TEXTLIST OutputText
  0 = 'OUT00 三色灯红' | Chinese: 'OUT00 三色灯红' | English: 'OUT00 Beacon_Red' | Vietnamese: 'OUT00 ?èn ?? ba màu ?'
  1 = 'OUT01 三色灯黄' | Chinese: 'OUT01 三色灯黄' | English: 'OUT01 Beacon_Yellow' | Vietnamese: 'OUT01 ?èn màu vàng ?'
  2 = 'OUT02 三色灯绿' | Chinese: 'OUT02 三色灯绿' | English: 'OUT02 Beacon_Green' | Vietnamese: 'OUT02 Màu xanh lá c?y ?èn ba màu ?'
  3 = 'OUT03 蜂鸣器' | Chinese: 'OUT03 蜂鸣器' | English: 'OUT03 Beacon_Buzzer' | Vietnamese: 'OUT03 buzzer ?'
  4 = 'OUT04 运行指示灯' | Chinese: 'OUT04 运行指示灯' | English: 'OUT04 Runing' | Vietnamese: 'OUT04 Ch?y ánh sáng ?'
  5 = 'OUT05 停止指示灯' | Chinese: 'OUT05 停止指示灯' | English: 'OUT05 Stop' | Vietnamese: 'OUT05 D?ng ?èn ?'
  6 = 'OUT06 照明灯' | Chinese: 'OUT06 照明灯' | English: 'OUT06 LED' | Vietnamese: 'OUT06 ?nh sáng ?'
  7 = 'OUT07 预留' | Chinese: 'OUT07 预留' | English: 'OUT07 None1' | Vietnamese: 'OUT07 Dành riêng ?'
  8 = 'OUT08 解锁站解压侧推气缸到原位' | Chinese: 'OUT08 解锁站解压侧推气缸到原位' | English: 'OUT08 OpenLockPressPush_Cyl_H' | Vietnamese: 'OUT08 OpenLockPressPush_Cyl_H'
  9 = 'OUT09 解锁站解压侧推气缸到工作位' | Chinese: 'OUT09 解锁站解压侧推气缸到工作位' | English: 'OUT09 OpenLockPressPush_Cyl_W' | Vietnamese: 'OUT09 OpenLockPressPush_Cyl_W'
  10 = 'OUT0A 解锁站解压旋转气缸到原位' | Chinese: 'OUT0A 解锁站解压旋转气缸到原位' | English: 'OUT0A OpenLockPressRotate_Cyl_H' | Vietnamese: 'OUT0A OpenLockPressRotate_Cyl_H'
  11 = 'OUT0B 解锁站解压旋转气缸到工作位' | Chinese: 'OUT0B 解锁站解压旋转气缸到工作位' | English: 'OUT0B OpenLockPressRotate_Cyl_W' | Vietnamese: 'OUT0B OpenLockPressRotate_Cyl_W'
  12 = 'OUT0C 主流线拨料升降气缸到原位' | Chinese: 'OUT0C 主流线拨料升降气缸到原位' | English: 'OUT0C Line0PushElevator_Cyl_H' | Vietnamese: 'OUT0C Line0PushElevator_Cyl_H'
  13 = 'OUT0D 主流线拨料升降气缸到工作位' | Chinese: 'OUT0D 主流线拨料升降气缸到工作位' | English: 'OUT0D Line0PushElevator_Cyl_W' | Vietnamese: 'OUT0D Line0PushElevator_Cyl_W'
  14 = 'OUT0E 接驳线前前阻挡气缸缩回' | Chinese: 'OUT0E 接驳线前前阻挡气缸缩回' | English: 'OUT0E AcquirePrevent2_Cyl_H' | Vietnamese: 'OUT0E AcquirePrevent2_Cyl_H'
  15 = 'OUT0F 接驳线前前阻挡气缸伸出' | Chinese: 'OUT0F 接驳线前前阻挡气缸伸出' | English: 'OUT0F AcquirePrevent2_Cyl_W' | Vietnamese: 'OUT0F AcquirePrevent2_Cyl_W'
  16 = 'OUT10 主流线分料气缸缩回' | Chinese: 'OUT10 主流线分料气缸缩回' | English: 'OUT10 Line0Part_Cyl_H' | Vietnamese: 'OUT10 Xi lanh c?a dòng chính rút lui ?'
  17 = 'OUT11 主流线分料气缸伸出' | Chinese: 'OUT11 主流线分料气缸伸出' | English: 'OUT11 Line0Part_Cyl_W' | Vietnamese: 'OUT11 Xi lanh dòng chính ra ngoài ?'
  18 = 'OUT12 主流线阻挡气缸缩回' | Chinese: 'OUT12 主流线阻挡气缸缩回' | English: 'OUT12 Line0Prevent_Cyl_H' | Vietnamese: 'OUT12 Dòng chính ng?n ch?n s? rút l?i c?a xi lanh ?'
  19 = 'OUT13 主流线阻挡气缸伸出' | Chinese: 'OUT13 主流线阻挡气缸伸出' | English: 'OUT13 Line0Prevent_Cyl_W' | Vietnamese: 'OUT13 Dòng chính ng?n các xi lanh thoát ra ?'
  20 = 'OUT14 主流线拨料气缸缩回' | Chinese: 'OUT14 主流线拨料气缸缩回' | English: 'OUT14 Line0Push_Cyl_H' | Vietnamese: 'OUT14 Xi lanh quay dòng chính rút lui ?'
  21 = 'OUT15 主流线拨料气缸伸出' | Chinese: 'OUT15 主流线拨料气缸伸出' | English: 'OUT15 Line0Push_Cyl_W' | Vietnamese: 'OUT15 Xi lanh cu?n dòng chính thò ra ?'
  22 = 'OUT16 接驳线前阻挡气缸缩回' | Chinese: 'OUT16 接驳线前阻挡气缸缩回' | English: 'OUT16 AcquirePrevent0_Cyl_H' | Vietnamese: 'OUT16 Khóa xi lanh tr??c d?y n?i rút l?i ?'
  23 = 'OUT17 接驳线前阻挡气缸伸出' | Chinese: 'OUT17 接驳线前阻挡气缸伸出' | English: 'OUT17 AcquirePrevent0_Cyl_W' | Vietnamese: 'OUT17 Ch?n xi lanh tr??c d?y n?i ?'
  24 = 'OUT18 接驳线后阻挡气缸缩回' | Chinese: 'OUT18 接驳线后阻挡气缸缩回' | English: 'OUT18 AcquirePrevent1_Cyl_H' | Vietnamese: 'OUT18 Khóa xi lanh l?i sau khi k?t n?i ?'
  25 = 'OUT19 接驳线后阻挡气缸伸出' | Chinese: 'OUT19 接驳线后阻挡气缸伸出' | English: 'OUT19 AcquirePrevent1_Cyl_W' | Vietnamese: 'OUT19 Ch?n xi lanh ra sau d?y n?i ?'
  26 = 'OUT1A 接驳线顶升气缸缩回' | Chinese: 'OUT1A 接驳线顶升气缸缩回' | English: 'OUT1A AcquireLift_Cyl_H' | Vietnamese: 'OUT1A Xi lanh n?ng d?y n?i rút l?i ?'
  27 = 'OUT1B 接驳线顶升气缸伸出' | Chinese: 'OUT1B 接驳线顶升气缸伸出' | English: 'OUT1B AcquireLift_Cyl_W' | Vietnamese: 'OUT1B Xi lanh c?m trên d?y d?n ra ngoài ?'
  28 = 'OUT1C 接驳模组拨料气缸缩回' | Chinese: 'OUT1C 接驳模组拨料气缸缩回' | English: 'OUT1C AcquirePush_Cyl_H' | Vietnamese: 'OUT1C Xi lanh k?t n?i m?-?un quay l?i ?'
  29 = 'OUT1D 接驳模组拨料气缸伸出' | Chinese: 'OUT1D 接驳模组拨料气缸伸出' | English: 'OUT1D AcquirePush_Cyl_W' | Vietnamese: 'OUT1D Xi lanh k?t n?i m?-?un phát ra ?'
  30 = 'OUT1E 接驳模组升降气缸缩回' | Chinese: 'OUT1E 接驳模组升降气缸缩回' | English: 'OUT1E AcquireElevator_Cyl_H' | Vietnamese: 'OUT1E Xi lanh n?ng m?-?un n?i rút l?i ?'
  31 = 'OUT1F 接驳模组升降气缸伸出' | Chinese: 'OUT1F 接驳模组升降气缸伸出' | English: 'OUT1F AcquireElevator_Cyl_W' | Vietnamese: 'OUT1F Xi lanh n?ng m?-?un n?i thò ra ?'
  32 = 'OUT20 转向站顶升气缸缩回' | Chinese: 'OUT20 转向站顶升气缸缩回' | English: 'OUT20 SteeringLift_Cyl_H' | Vietnamese: 'OUT20 Quay tr? l?i xi lanh ?'
  33 = 'OUT21 转向站顶升气缸伸出' | Chinese: 'OUT21 转向站顶升气缸伸出' | English: 'OUT21 SteeringLift_Cyl_W' | Vietnamese: 'OUT21 Các xi lanh m? ra ?'
  34 = 'OUT22 转向站接驳升降气缸缩回' | Chinese: 'OUT22 转向站接驳升降气缸缩回' | English: 'OUT22 SteeringAcquireElevator_Cyl_H' | Vietnamese: 'OUT22 Quay l?i v?i xi lanh n?ng t?i tr?m lái ?'
  35 = 'OUT23 转向站接驳升降气缸伸出' | Chinese: 'OUT23 转向站接驳升降气缸伸出' | English: 'OUT23 SteeringAcquireElevator_Cyl_W' | Vietnamese: 'OUT23 Các xi lanh n?ng ???c n?i v?i các tr?m r? ?'
  36 = 'OUT24 转向站旋转气缸缩回' | Chinese: 'OUT24 转向站旋转气缸缩回' | English: 'OUT24 SteeringRotate_Cyl_H' | Vietnamese: 'OUT24 Quay tr?m quay xi lanh ?? rút lui ?'
  37 = 'OUT25 转向站旋转气缸伸出' | Chinese: 'OUT25 转向站旋转气缸伸出' | English: 'OUT25 SteeringRotate_Cyl_W' | Vietnamese: 'OUT25 Các xi lanh xoay ? v? trí quay thò ra ?'
  38 = 'OUT26 转向站接驳限位气缸缩回' | Chinese: 'OUT26 转向站接驳限位气缸缩回' | English: 'OUT26 SteeringAcquireLimit_Cyl_H' | Vietnamese: 'OUT26 Quay l?i xi lanh gi?i h?n k?t n?i tr?m r? ?'
  39 = 'OUT27 转向站接驳限位气缸伸出' | Chinese: 'OUT27 转向站接驳限位气缸伸出' | English: 'OUT27 SteeringAcquireLimit_Cyl_W' | Vietnamese: 'OUT27 Xi lanh gi?i h?n k?t n?i v?i tr?m lái xe ???c thò ra ?'
  40 = 'OUT28 解锁站阻挡气缸缩回' | Chinese: 'OUT28 解锁站阻挡气缸缩回' | English: 'OUT28 OpenLockPrevent_Cyl_H' | Vietnamese: 'OUT28 Tr?m m? khóa ng?n ch?n s? rút lui xi lanh ?'
  41 = 'OUT29 解锁站阻挡气缸伸出' | Chinese: 'OUT29 解锁站阻挡气缸伸出' | English: 'OUT29 OpenLockPrevent_Cyl_W' | Vietnamese: 'OUT29 Tr?m m? khóa ng?n ch?n các xi lanh thò ra ?'
  42 = 'OUT2A 解锁站顶升气缸缩回' | Chinese: 'OUT2A 解锁站顶升气缸缩回' | English: 'OUT2A OpenLockLift_Cyl_H' | Vietnamese: 'OUT2A M? khóa tr?m n?ng xi lanh rút lui ?'
  43 = 'OUT2B 解锁站顶升气缸伸出' | Chinese: 'OUT2B 解锁站顶升气缸伸出' | English: 'OUT2B OpenLockLift_Cyl_W' | Vietnamese: 'OUT2B Xi lanh m? khóa tr? n?ng thò ra ?'
  44 = 'OUT2C 解锁站侧推气缸缩回' | Chinese: 'OUT2C 解锁站侧推气缸缩回' | English: 'OUT2C OpenLockPush_Cyl_H' | Vietnamese: 'OUT2C M? khóa các xi lanh ??y ga ?? rút lui ?'
  45 = 'OUT2D 解锁站侧推气缸伸出' | Chinese: 'OUT2D 解锁站侧推气缸伸出' | English: 'OUT2D OpenLockPush_Cyl_W' | Vietnamese: 'OUT2D M? khóa ga ??y xi lanh thò ra ?'
  46 = 'OUT2E 解锁站旋转气缸缩回' | Chinese: 'OUT2E 解锁站旋转气缸缩回' | English: 'OUT2E OpenLockRotate_Cyl_H' | Vietnamese: 'OUT2E M? khóa tr?m quay xi lanh rút lui ?'
  47 = 'OUT2F 解锁站旋转气缸伸出' | Chinese: 'OUT2F 解锁站旋转气缸伸出' | English: 'OUT2F OpenLockRotate_Cyl_W' | Vietnamese: 'OUT2F Xi lanh xoay ? v? trí m? khóa thò ra ?'
  48 = 'OUT30 解锁站侧推气缸2缩回' | Chinese: 'OUT30 解锁站侧推气缸2缩回' | English: 'OUT30 OpenLockPush2_Cyl_H' | Vietnamese: 'OUT30 M? khóa ga bên ??y xi lanh 2 rút lui ?'
  49 = 'OUT31 解锁站侧推气缸2伸出' | Chinese: 'OUT31 解锁站侧推气缸2伸出' | English: 'OUT31 OpenLockPush2_Cyl_W' | Vietnamese: 'OUT31 M? khóa ga ??y xi lanh 2 thò ra ?'
  50 = 'OUT32 取UC站阻挡气缸缩回' | Chinese: 'OUT32 取UC站阻挡气缸缩回' | English: 'OUT32 TakeUcPrevent_Cyl_H' | Vietnamese: 'OUT32 L?y các tr?m ng?n ch?n và rút l?i xi lanh ?'
  51 = 'OUT33 取UC站阻挡气缸伸出' | Chinese: 'OUT33 取UC站阻挡气缸伸出' | English: 'OUT33 TakeUcPrevent_Cyl_W' | Vietnamese: 'OUT33 L?y ga ng?n ch?n lít ra ?'
  52 = 'OUT34 取UC站顶升气缸缩回' | Chinese: 'OUT34 取UC站顶升气缸缩回' | English: 'OUT34 TakeUcLift_Cyl_H' | Vietnamese: 'OUT34 L?y xi lanh n?ng lên c?a tr?m UC và rút lui ?'
  53 = 'OUT35 取UC站顶升气缸伸出' | Chinese: 'OUT35 取UC站顶升气缸伸出' | English: 'OUT35 TakeUcLift_Cyl_W' | Vietnamese: 'OUT35 L?y xi lanh n?ng lên t? tr?m UC ?'
  54 = 'OUT36 取UC站侧推气缸缩回' | Chinese: 'OUT36 取UC站侧推气缸缩回' | English: 'OUT36 TakeUcPush_Cyl_H' | Vietnamese: 'OUT36 L?y xi lanh ??y bên tàu và rút lui ?'
  55 = 'OUT37 取UC站侧推气缸伸出' | Chinese: 'OUT37 取UC站侧推气缸伸出' | English: 'OUT37 TakeUcPush_Cyl_W' | Vietnamese: 'OUT37 L?y ga bên ??y ra kh?i xi lanh ?'
  56 = 'OUT38 取UC站旋转气缸缩回' | Chinese: 'OUT38 取UC站旋转气缸缩回' | English: 'OUT38 TakeUcRotate_Cyl_H' | Vietnamese: 'OUT38 L?y xi lanh quay ? tr?m UC và rút lui ?'
  57 = 'OUT39 取UC站旋转气缸伸出' | Chinese: 'OUT39 取UC站旋转气缸伸出' | English: 'OUT39 TakeUcRotate_Cyl_W' | Vietnamese: 'OUT39 L?y các xi lanh quay t? tr?m UC ?'
  58 = 'OUT3A 取UC站校平气缸原位' | Chinese: 'OUT3A 取UC站校平气缸原位' | English: 'OUT3A TakeUcStandard_Cyl_H' | Vietnamese: 'OUT3A L?y xi lanh ph?ng ? ga UC ?'
  59 = 'OUT3B 取UC站校平气缸工作位' | Chinese: 'OUT3B 取UC站校平气缸工作位' | English: 'OUT3B TakeUcStandard_Cyl_W' | Vietnamese: 'OUT3B Tr?m ki?m tra xi lanh b?ng ph?ng ?'
  60 = 'OUT3C 取UC站工装夹紧气缸原位' | Chinese: 'OUT3C 取UC站工装夹紧气缸原位' | English: 'OUT3C TakeUcFrockClamp_Cyl_H' | Vietnamese: 'OUT3C L?y xi lanh k?p vào v? trí c?a tr?m UC'
  61 = 'OUT3D 取UC站工装夹紧气缸工作位' | Chinese: 'OUT3D 取UC站工装夹紧气缸工作位' | English: 'OUT3D TakeUcFrockClamp_Cyl_W' | Vietnamese: 'OUT3D L?y v? trí làm vi?c xi lanh cài ??t ? ga UC'
  62 = 'OUT3E 下工装站阻挡气缸缩回' | Chinese: 'OUT3E 下工装站阻挡气缸缩回' | English: 'OUT3E UnloadFrockPrevent_Cyl_H' | Vietnamese: 'OUT3E Ng?n ch?n các xi lanh rút lui ?'
  63 = 'OUT3F 下工装站阻挡气缸伸出' | Chinese: 'OUT3F 下工装站阻挡气缸伸出' | English: 'OUT3F UnloadFrockPrevent_Cyl_W' | Vietnamese: 'OUT3F Ng?n ch?n các xi lanh ra ngoài ?'
  64 = 'OUT40 下工装站顶升气缸缩回' | Chinese: 'OUT40 下工装站顶升气缸缩回' | English: 'OUT40 UnloadFrockLift_Cyl_H' | Vietnamese: 'OUT40 Xi lanh n?ng xu?ng ga xu?ng rút lui ?'
  65 = 'OUT41 下工装站顶升气缸伸出' | Chinese: 'OUT41 下工装站顶升气缸伸出' | English: 'OUT41 UnloadFrockLift_Cyl_W' | Vietnamese: 'OUT41 Xi lanh n?ng lên t? tr?m t?i xu?ng ?'
  66 = 'OUT42 下工装站拨料气缸缩回' | Chinese: 'OUT42 下工装站拨料气缸缩回' | English: 'OUT42 UnloadFrockPush_Cyl_H' | Vietnamese: 'OUT42 Xi lanh xi lanh quay tr? l?i tr?m t?i xu?ng ?'
  67 = 'OUT43 下工装站拨料气缸伸出' | Chinese: 'OUT43 下工装站拨料气缸伸出' | English: 'OUT43 UnloadFrockPush_Cyl_W' | Vietnamese: 'OUT43 Xi lanh ngu?n l?c ti?p theo ?'
  68 = 'OUT44 取UC模组平移Y气缸缩回' | Chinese: 'OUT44 取UC模组平移Y气缸缩回' | English: 'OUT44 TakeUc1Y_Cyl_H' | Vietnamese: 'OUT44 L?y m?-?un UC chuy?n xi lanh Y và rút lui ?'
  69 = 'OUT45 取UC模组平移Y气缸伸出' | Chinese: 'OUT45 取UC模组平移Y气缸伸出' | English: 'OUT45 TakeUc1Y_Cyl_W' | Vietnamese: 'OUT45 L?y m?-?un UC và di chuy?n xi lanh Y ra ngoài ?'
  70 = 'OUT46 取UC模组升降Z1气缸缩回' | Chinese: 'OUT46 取UC模组升降Z1气缸缩回' | English: 'OUT46 TakeUc1Z1_Cyl_H' | Vietnamese: 'OUT46 L?y m?-?un UC n?ng xi lanh Z1 ?? rút lui ?'
  71 = 'OUT47 取UC模组升降Z1气缸伸出' | Chinese: 'OUT47 取UC模组升降Z1气缸伸出' | English: 'OUT47 TakeUc1Z1_Cyl_W' | Vietnamese: 'OUT47 N?ng xi lanh ra kh?i m?-?un UC ?'
  72 = 'OUT48 取UC模组升降Z2气缸缩回' | Chinese: 'OUT48 取UC模组升降Z2气缸缩回' | English: 'OUT48 TakeUc1Z2_Cyl_H' | Vietnamese: 'OUT48 L?y m?-?un UC n?ng xi lanh Z2 ?? rút lui ?'
  73 = 'OUT49 取UC模组升降Z2气缸伸出' | Chinese: 'OUT49 取UC模组升降Z2气缸伸出' | English: 'OUT49 TakeUc1Z2_Cyl_W' | Vietnamese: 'OUT49 ??a ?ng n?ng Z2 ra kh?i m?-?un UC ?'
  74 = 'OUT4A 取UC模组旋转气缸缩回' | Chinese: 'OUT4A 取UC模组旋转气缸缩回' | English: 'OUT4A TakeUc1Rotate_Cyl_H' | Vietnamese: 'OUT4A Thu h?i xi lanh quay b?ng m?-?un UC ?'
  75 = 'OUT4B 取UC模组旋转气缸伸出' | Chinese: 'OUT4B 取UC模组旋转气缸伸出' | English: 'OUT4B TakeUc1Rotate_Cyl_W' | Vietnamese: 'OUT4B L?y m?-?un UC xoay xi lanh ra ngoài ?'
  76 = 'OUT4C 取UC模组夹紧气缸缩回' | Chinese: 'OUT4C 取UC模组夹紧气缸缩回' | English: 'OUT4C TakeUc1Clamp_Cyl_H' | Vietnamese: 'OUT4C L?y m?-?un UC k?p xi lanh ?? rút lui ?'
  77 = 'OUT4D 取UC模组夹紧气缸伸出' | Chinese: 'OUT4D 取UC模组夹紧气缸伸出' | English: 'OUT4D TakeUc1Clamp_Cyl_W' | Vietnamese: 'OUT4D L?y m?-?un và k?p ?ng ra ?'
  78 = 'OUT4E 下UC皮带升降气缸缩回' | Chinese: 'OUT4E 下UC皮带升降气缸缩回' | English: 'OUT4E UnloadUcElevator_Cyl_H' | Vietnamese: 'OUT4E Thu h?i xi lanh n?ng d??i vành ?ai UC ?'
  79 = 'OUT4F 下UC皮带升降气缸伸出' | Chinese: 'OUT4F 下UC皮带升降气缸伸出' | English: 'OUT4F UnloadUcElevator_Cyl_W' | Vietnamese: 'OUT4F Xi lanh n?ng d??i vành ?ai UC thò ra ?'
  80 = 'OUT50 下UC皮带拨料气缸缩回' | Chinese: 'OUT50 下UC皮带拨料气缸缩回' | English: 'OUT50 UnloadUcConveyorPush_Cyl_H' | Vietnamese: 'OUT50 Quay l?i xi lanh quay d??i vành ?ai UC ?'
  81 = 'OUT51 下UC皮带拨料气缸伸出' | Chinese: 'OUT51 下UC皮带拨料气缸伸出' | English: 'OUT51 UnloadUcConveyorPush_Cyl_W' | Vietnamese: 'OUT51 Cái xi lanh d??i vành ?ai UC thò ra ?'
  82 = 'OUT52 下工装皮带升降气缸缩回' | Chinese: 'OUT52 下工装皮带升降气缸缩回' | English: 'OUT52 UnloadFrockConveyorPrevent_Cyl_H' | Vietnamese: 'OUT52 Th?t l?ng n?ng xi lanh kéo xu?ng ?'
  83 = 'OUT53 下工装皮带升降气缸伸出' | Chinese: 'OUT53 下工装皮带升降气缸伸出' | English: 'OUT53 UnloadFrockConveyorPrevent_Cyl_W' | Vietnamese: 'OUT53 Xi lanh n?ng vành ?ai c?ng vi?c thò ra ?'
  84 = 'OUT54 下工装皮带拨料气缸缩回' | Chinese: 'OUT54 下工装皮带拨料气缸缩回' | English: 'OUT54 UnloadFrockConveyorPush_Cyl_H' | Vietnamese: 'OUT54 ?óng gói vành ?ai xi lanh quay l?i ?'
  85 = 'OUT55 下工装皮带拨料气缸伸出' | Chinese: 'OUT55 下工装皮带拨料气缸伸出' | English: 'OUT55 UnloadFrockConveyorPush_Cyl_W' | Vietnamese: 'OUT55 Xi lanh vành ?ai c?ng c? thò ra ?'
  86 = 'OUT56 接驳线前步进' | Chinese: 'OUT56 接驳线前步进' | English: 'OUT56 AcquireFrontAxis' | Vietnamese: 'OUT56 AcquireFrontAxis'
  87 = 'OUT57 接驳线步进' | Chinese: 'OUT57 接驳线步进' | English: 'OUT57 AcquireAxis' | Vietnamese: 'OUT57 B??c trên d?y n?i ?'
  88 = 'OUT58 拆解线步进' | Chinese: 'OUT58 拆解线步进' | English: 'OUT58 DismantlingAxis' | Vietnamese: 'OUT58 B??c c?t d?y ?'
  89 = 'OUT59 下UC皮带步进' | Chinese: 'OUT59 下UC皮带步进' | English: 'OUT59 UnloadUcAxis' | Vietnamese: 'OUT59 B??c xu?ng d??i vành ?ai UC ?'
  90 = 'OUT5A 下工装皮带步进' | Chinese: 'OUT5A 下工装皮带步进' | English: 'OUT5A UnloadFrock' | Vietnamese: 'OUT5A D?y n?t di chuy?n ?'
  91 = 'OUT5B 预留' | Chinese: 'OUT5B 预留' | English: 'OUT5B None21' | Vietnamese: 'OUT5B Dành riêng ?'
  92 = 'OUT5C 下UC皮带翻转气缸缩回' | Chinese: 'OUT5C 下UC皮带翻转气缸缩回' | English: 'OUT5C UnloadUcBeltTipper_Cyl_H' | Vietnamese: 'OUT5C Quay ng??c xi lanh l?i ?'
  93 = 'OUT5D 下UC皮带翻转气缸伸出' | Chinese: 'OUT5D 下UC皮带翻转气缸伸出' | English: 'OUT5D UnloadUcBeltTipper_Cyl_W' | Vietnamese: 'OUT5D Cái xi lanh xoay d??i vành ?ai UC thò ra ?'
  94 = 'OUT5E 下UC皮带顶升气缸缩回' | Chinese: 'OUT5E 下UC皮带顶升气缸缩回' | English: 'OUT5E UnloadUcBeltLift_Cyl_H' | Vietnamese: 'OUT5E Co l?i xi lanh n?ng lên d??i vành ?ai UC ?'
  95 = 'OUT5F 下UC皮带顶升气缸伸出' | Chinese: 'OUT5F 下UC皮带顶升气缸伸出' | English: 'OUT5F UnloadUcBeltLift_Cyl_W' | Vietnamese: 'OUT5F Cái xi lanh n?ng lên d??i vành ?ai UC thò ra ?'
  96 = 'OUT60 解锁站升降气缸原位' | Chinese: 'OUT60 解锁站升降气缸原位' | English: 'OUT60 OpenLockElevator_Cyl_H' | Vietnamese: 'OUT60 M? khóa tr?m n?ng xi lanh v? trí ?'
  97 = 'OUT61 解锁站升降气缸工作位' | Chinese: 'OUT61 解锁站升降气缸工作位' | English: 'OUT61 OpenLockElevator_Cyl_W' | Vietnamese: 'OUT61 M? khóa tr?m n?ng xi lanh v? trí làm vi?c ?'
  98 = 'OUT62 解锁站解锁平移原位' | Chinese: 'OUT62 解锁站解锁平移原位' | English: 'OUT62 OpenLockTranslation_Cyl_H' | Vietnamese: 'OUT62 Tr?m m? khóa m? khóa chuy?n v? trí ?'
  99 = 'OUT63 解锁站解锁平移工作位' | Chinese: 'OUT63 解锁站解锁平移工作位' | English: 'OUT63 OpenLockTranslation_Cyl_W' | Vietnamese: 'OUT63 Tr?m m? khóa m? khóa chuy?n v? trí làm vi?c ?'
  100 = 'OUT64 解锁站按压气缸到原位' | Chinese: 'OUT64 解锁站按压气缸到原位' | English: 'OUT64 OpenLockPin_Cyl_H' | Vietnamese: 'OUT64 M? khóa tr?m nh?n xi lanh vào v? trí ?'
  101 = 'OUT65 解锁站按压气缸到工作位' | Chinese: 'OUT65 解锁站按压气缸到工作位' | English: 'OUT65 OpenLockPin_Cyl_W' | Vietnamese: 'OUT65 M? khóa tr?m nh?n xi lanh ??n v? trí làm vi?c ?'
  102 = 'OUT66 取UC站升降气缸原位' | Chinese: 'OUT66 取UC站升降气缸原位' | English: 'OUT66 TakeUcElevator_Cyl_H' | Vietnamese: 'OUT66 L?y xi lanh n?ng t? tr?m UC ?'
  103 = 'OUT67 取UC站升降气缸工作位' | Chinese: 'OUT67 取UC站升降气缸工作位' | English: 'OUT67 TakeUcElevator_Cyl_W' | Vietnamese: 'OUT67 Tr? UC n?ng xi lanh v? trí làm vi?c ?'
  104 = 'OUT68 取UC站侧推1气缸到原位' | Chinese: 'OUT68 取UC站侧推1气缸到原位' | English: 'OUT68 TakeUcPush1_Cyl_H' | Vietnamese: 'OUT68 L?y ga UC ??y 1 xi lanh vào v? trí ?'
  105 = 'OUT69 取UC站侧推1气缸到工作位' | Chinese: 'OUT69 取UC站侧推1气缸到工作位' | English: 'OUT69 TakeUcPush1_Cyl_W' | Vietnamese: 'OUT69 L?y ga bên ??y 1 xi lanh t?i v? trí làm vi?c ?'
  106 = 'OUT6A 预留' | Chinese: 'OUT6A 预留' | English: 'OUT6A None35' | Vietnamese: 'OUT6A Dành riêng ?'
  107 = 'OUT6B 预留' | Chinese: 'OUT6B 预留' | English: 'OUT6B None36' | Vietnamese: 'OUT6B Dành riêng ?'
  108 = 'OUT6C 预留' | Chinese: 'OUT6C 预留' | English: 'OUT6C None37' | Vietnamese: 'OUT6C Dành riêng ?'
  109 = 'OUT6D 预留' | Chinese: 'OUT6D 预留' | English: 'OUT6D None38' | Vietnamese: 'OUT6D Dành riêng ?'
  110 = 'OUT6E 预留' | Chinese: 'OUT6E 预留' | English: 'OUT6E None39' | Vietnamese: 'OUT6E Dành riêng ?'
  111 = 'OUT6F 预留' | Chinese: 'OUT6F 预留' | English: 'OUT6F None40' | Vietnamese: 'OUT6F Dành riêng ?'
   = ''
END_TEXTLIST

(* stored: Version 1.1.0.1, ProductVersion 3.1.4024.3
   TextList OutputText: Id {3e72ff28-dbe1-48a8-be85-75c7936f53c1} *)
